// TIA Portal V20 export
DATA_BLOCK "DB_AxisPosMachineNC"   // DB82
{ S7_Optimized_Access := 'TRUE' }
// stored: MemoryReserve 100
   VAR
      Axis_X : Struct
         Load : LReal := 249.3;
         Unload : LReal := 324.5;
         Blowing : LReal := 287.3;
      END_STRUCT;
      Axis_Y : Struct
         Load : LReal := 55.02;
         Unload : LReal := 55.02;
         Blowing : LReal := 55.02;
      END_STRUCT;
      Axis_B : Struct
         Load : LReal := 0.0;
         Unload : LReal := 0.0;
         Blowing : LReal := 0.0;
      END_STRUCT;
      Axis_ZM : Struct
         Safe : Real := 145.0;
      END_STRUCT;
      Axis_ZL : Struct
         Safe : Real := 14.0;
      END_STRUCT;
   END_VAR
BEGIN
END_DATA_BLOCK
